{attribute 'pack_mode' := '1'}
TYPE MoveAxisAbsolute EXTENDS IncomingMessage :
STRUCT
	axisIndex: INT; (* 1 or 2.*)
	position: LREAL;
	speed: LREAL;
END_STRUCT
END_TYPE

(* stored: Version 1.1.0.1, ProductVersion 3.1.4022.12
   DUT MoveAxisAbsolute: Id {ad3159c0-09d6-42dc-904b-0cbebc62be45} *)
